// TIA Portal V20 export
DATA_BLOCK "T4 LANT I-O"   // DB1612
{ S7_Optimized_Access := 'TRUE' }
AUTHOR : SAS
// stored: AutoNumber false, IsRetainMemResEnabled true, MemoryReserve 100, RetainMemoryReserve 100
   VAR
      DI : Struct
         "T4-B49.X1" : Bool;   // (E0.3) T4-Senzor Proximitate Pozitia "Incetinire" 1
         "T4-B49.X2" : Bool;   // (E0.4) T4-Senzor Proximitate Pozitia "Incetinire" 2
         "S45.1" : Bool;   // (E79.0) T4 Lant Comanda 'Inainte'
         "S45.2" : Bool;   // (E79.1) T4 Lant Comanda 'Inapoi'
         "S45.3" : Bool;   // (E79.2) T4 Lant Selectie 'Pas/Continuu'
         "S45.4" : Bool;   // (E79.3) T4 Lant Rostogolire Comanda Inainte
         "S45.5" : Bool;   // (E79.4) T4 Lant Rostogolire Comanda Inapoi
         "B48.5" : Bool;   // (E81.4) T4 Lant Senzor 1 Prezenta Teava pe Lant (intrare)
         "B48.6" : Bool;   // (E81.5) T4 Lant Senzor 2 Prezenta Teava pe Lant (intrare)
         "B48.7" : Bool;   // (E81.6) T4 Lant Senzor 'Pas'
         "E81.7" : Bool;   // (E81.7) T4 senzor1 suplimentar la tevi scurte
         "B49.1" : Bool;   // (E82.0) T4 Lant Senzor 1 Prezenta Teava pe Lant(pendula opritor iesire)
         "B49.2" : Bool;   // (E82.1) T4 Lant Senzor 2 Prezenta Teava pe Lant (pendula opritor iesire)
         "Q21.2/K21.2" : Bool;   // (E214.0) T4 Lant Tensiune Comanda
         "Q11.7" : Bool;   // (E215.0) T4 Lant Disjunctor Alimentare Ventilatoare Motoare
         "Q11.3" : Bool;   // (E215.1) T4 Lant Disjunctor Alimentare Convertizor
         "K22.2no" : Bool;   // (E215.2) T4 Lant Confirmare Cuplare Contactor Convertizor
         "K22.6no" : Bool;   // (E215.3) T4 Lant Confirmare Cuplare Contactor Frana
         "K24.5.1" : Bool;   // (E215.4) T4 Lant Convertizor 'OK'
         "K24.5.2" : Bool;   // (E215.5) T4 Lant Convertizor 'RUN'
         "S33.7" : Bool;   // (E215.6) T4 Lant Permisie Cuplare Contactor
         "Q11.8" : Bool;   // (E215.7) T4 Lant Disjunctor Alimentare Frana
         "Q17.3" : Bool;   // (E217.1) T4 Lant Rostogolire Disjunctor Alimentare Convertizor
         "K26.2no" : Bool;   // (E217.2) T4 Lant Rostogolire Confirmare Cuplare Contactor Convertizor
         "U17.3'OK'" : Bool;   // (E217.4) T4 Lant Rostogolire Convertizor 'OK'
         "U17.3(RUN)" : Bool;   // (E217.5) T4 Lant Rostogolire Convertizor 'RUN'
         "S35.7" : Bool;   // (E217.6) T4 Lant Rostogolire Permisie Cuplare Contactor
         "F17.3" : Bool;   // (E217.7) T4 Lant Rostogolire Protectie Termica Motor
      END_STRUCT;
      "DO" : Struct
         "K52.7-K22.6" : Bool;   // (A190.6) T4 Lant Contactor Frana
         "K54.5" : Bool;   // (A191.4) T4 Lant Rostogolire Contactor Alimentare Convertizor
         "K54.6" : Bool;   // (A191.5) T4 Lant Rostogolire Contactor 'Abilitare'
         "A191.6" : Bool;   // (A191.6) Ventilator racire motor rostogolire
         "K55.5-K22.2" : Bool;   // (A200.4) T4 Lant Contactor Alimentare Convertizor
         "K55.6" : Bool;   // (A200.5) T4 Lant Contactor 'Abilitare'
         "K55.7" : Bool;   // (A200.6) T4 Lant Contactor Deplasare 'Inainte'
         "K55.8" : Bool;   // (A200.7) T4 Lant Contactor Deplasare 'Inapoi'
      END_STRUCT;
      "Drive Lant" : Struct
         CMD : "DRIVE_CMD_Horiz";
         STATUS { S7_SetPoint := 'True'} : "DRIVE_STATUS_Horiz";
         RD_AREA : "G120-Telegram1 READ";
         WR_AREA : "G120-Telegram1-WRITE";
      END_STRUCT;
      "Drive LantRost" : Struct
         CMD : "DRIVE_CMD_Horiz";
         STATUS { S7_SetPoint := 'True'} : "DRIVE_STATUS_Horiz";
         RD_AREA : "G120-Telegram352-Mod READ";
         WR_AREA : "G120-Telegram352-Mod WRITE";
      END_STRUCT;
   END_VAR
BEGIN
END_DATA_BLOCK
